(* CoDeSys 2.3.9.50 project: 4F.pr6 *)
(* Libraries: STANDARD.LB6 5.6.98 12:03:02 *)

(* POU MAIN, LD *)
PROGRAM MAIN
VAR
	Switch AT %IX0.0: BOOL;
	C1: CTU;
	Conveyer1Light AT %QX0.0: BOOL;
	C2: CTU;
	Motor AT %QX0.1: BOOL;
	A AT %QX0.5: BOOL;
	t1: TON;
END_VAR
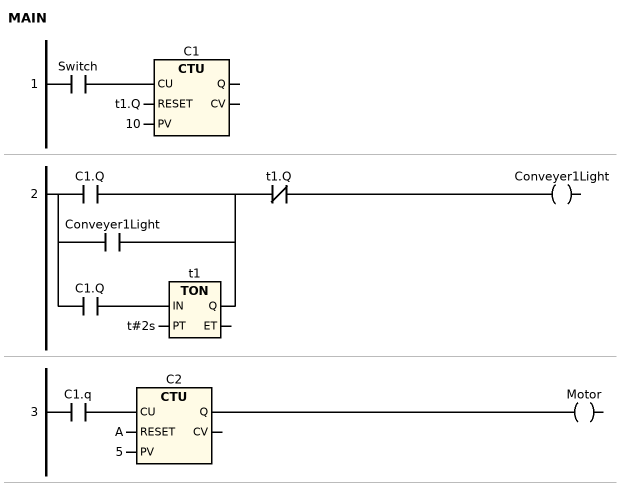
_LD_ (* Ladder Diagram *)
NETWORK 1
	[Switch] - C1:CTU(CU: *, RESET: t1.Q, PV: 10)
NETWORK 2
	{ [C1.Q] | [Conveyer1Light] | [C1.Q] - t1:TON(IN: *, PT: t#2s) } - [/t1.Q] --- (Conveyer1Light)
NETWORK 3
	[C1.q] - C2:CTU(CU: *, RESET: A, PV: 5) --- (Motor)
_END_LD_
(* the same logic as Structured Text *)
(* Network 1 *)
C1(CU := Switch, RESET := t1.Q, PV := 10);
(* Network 2 *)
t1(IN := C1.Q, PT := t#2s);
Conveyer1Light := (C1.Q OR Conveyer1Light OR t1.Q) AND NOT t1.Q;
(* Network 3 *)
C2(CU := C1.q, RESET := A, PV := 5);
Motor := C2.Q;
END_PROGRAM
